PROGRAM MAIN
VAR
	ESTACION: FB_Estacion;
END_VAR

ESTACION();

END_PROGRAM

(* stored: Version 1.1.0.1, ProductVersion 3.1.4024.12
   POU MAIN: Id {3e745d66-bce5-4a4f-9c7e-78379eb25dba}, SpecialFunc None *)
